// TwinCAT 3 PLC project PLC_LaserMarking_K2P3
// ProgramVersion: 3.1.4023.0
// libraries:
//   Tc2_MC2, * (Beckhoff Automation GmbH)
//   Tc2_Standard, * (Beckhoff Automation GmbH)
//   Tc2_System, * (Beckhoff Automation GmbH)
//   Tc3_MC2_AdvancedHoming, * (Beckhoff Automation GmbH)
//   Tc3_Module, * (Beckhoff Automation GmbH)
// project tree:
//   DUTs/ eAuto_State_Macine.TcTLEO, eLM_State_Machine.TcTLEO, eManual_State_Machine.TcTLEO, eMarking_Types.TcTLEO, eMC_State_Machine.TcTLEO, eUniquenessMethos.TcTLEO
//   GVLs/ GVL_AxisParameters.TcGVL, GVL_GateWay.TcGVL, GVL_IO.TcGVL, GVL_LaserMarking_MC_Parameters.TcGVL, GVL_StateMachine.TcGVL
//   / PlcTask.TcTTO
//   POUs/Alarms/ Alarm_Display_ST.TcPOU, Alarm_Flag.TcPOU, EtherCAT_Diagnostic.TcPOU
//   POUs/Main POUs/ Main.TcPOU, POU_GatewaySignals.TcPOU, POU_Manual_Auto.TcPOU, POU_Output.TcPOU
//   POUs/StateMachine_AutoManual/ AutoStates_POU.TcPOU
//   POUs/StateMachine_LaserMarking/ LaserMarking_Variable_Selection.TcPOU, LM_State_MC_TCP.TcPOU
//   POUs/StateMachine_MC_Axis/ MC_State_MC.TcPOU
// real-time tasks:
//   TASK PlcTask: cycle T#10ms, priority 20, ADS port 350
//   TASK PlcTask1: cycle T#10ms, priority 21, ADS port 351
// motion (NC):
//   TASK NC-Task SAF: cycle T#2ms, priority 4, ADS port 501
//   TASK NC-Task SVB: cycle T#10ms, priority 8, ADS port 511
//   AXIS Axis Y (id 2)
//     OtherSettings: AllowMotionCmdToSlave=true
//     encoder EncType=19
//       EncPara: MaxCount=#xffffffff
//     drive DrvType=16
//       DrvPara: MaxCount=#xffffffff, DriveControlDWord=#x00020000
//         Analog: TorqueScale=10, ScaleFactorActTorque=0.1
//         TimeComp: TaskDelayCycles=1
//     controller CtrType=1
//       CtrPara: PriorControlFactor=1
//         Observer: BandWidth=20
// I/O:
//   DEVICE Device 1 (EtherCAT), AmsNetId 192.168.0.10.2.1
//     Term 1 (EK1100) [EK1100 EtherCAT Coupler (2A E-Bus)]
//     Box 2 (ASDA-A2-E CoE Drive) [Delta ASDA-A2-E EtherCAT(CoE) Drive Rev4]
// variable links:
//   NC-Task SAF/Axes/Axis Y <-> Device 1 (EtherCAT)/Box 2 (ASDA-A2-E CoE Drive)
//     Drive/Inputs/In/nDcOutputTime <-> InfoData/DcOutputShift
//     Drive/Inputs/In/nState1 <-> 2nd TxPDO Mapping/Status Word
//     Drive/Inputs/In/nState2 <-> 2nd TxPDO Mapping/Status Word @bit 8
//     Drive/Inputs/In/nState4 @bit 1 <-> WcState/InputToggle
//     Drive/Inputs/In/nState4 <-> WcState/WcState
//     Drive/Outputs/Out/nCtrl1 <-> 2nd RxPDO Mapping/Control Word
//     Drive/Outputs/Out/nCtrl2 <-> 2nd RxPDO Mapping/Control Word @bit 8
//     Drive/Outputs/Out/nDataOut1 <-> 2nd RxPDO Mapping/TargetPosition
//     Enc/Inputs/In/nDataIn1 <-> 2nd TxPDO Mapping/ActualPosition
//     Enc/Inputs/In/nDcInputTime <-> InfoData/DcInputShift
//     Enc/Inputs/In/nState4 @bit 1 <-> WcState/InputToggle
//     Enc/Inputs/In/nState4 <-> WcState/WcState
//   PLC_LaserMarking_K2P3/PLC_LaserMarking_K2P3 Instance <-> NC-Task SAF/Axes/Axis Y
//     PlcTask Inputs/GVL_AxisParameters.YAxis.NcToPlc <-> Outputs/ToPlc
//     PlcTask Outputs/GVL_AxisParameters.YAxis.PlcToNc <-> Inputs/FromPlc

CONFIGURATION PLC_LaserMarking_K2P3
    RESOURCE PLC ON TwinCAT3
        TASK PlcTask(INTERVAL := T#10ms, PRIORITY := 21);
        PROGRAM Main WITH PlcTask : Main;
    END_RESOURCE
END_CONFIGURATION

// ---- DUTs/eAuto_State_Macine.TcTLEO
//{attribute 'qualified_only'}
{attribute 'strict'}
TYPE eAuto_State_Macine :
(
	Auto_Stop_State 	:= 0,
	Auto_Init_State 	:= 1,
	Auto_Ready_State 	:= 2,
	Auto_Y_Motion_State := 3,
	Auto_Marking_State 	:= 4
);
END_TYPE

// ---- DUTs/eLM_State_Machine.TcTLEO
//{attribute 'qualified_only'}
{attribute 'strict'}
TYPE eLM_State_Machine :
(
		LM_Off 			:= 0 ,
		LM_Init 		:= 1 ,
		LM_Ready 		:= 2 ,
		LM_CodeSend 	:= 3 ,
		LM_MarkCommand 	:= 4 ,
		LM_Feedback 	:= 5 
);
END_TYPE

// ---- DUTs/eManual_State_Machine.TcTLEO
//{attribute 'qualified_only'}
{attribute 'strict'}
TYPE eManual_State_Machine :
(
	Manual_Stop_State 	:= 0 ,
	Manual_Init_State 	:= 1 ,
	Manual_Ready_State 	:= 2 

);
END_TYPE

// ---- DUTs/eMarking_Types.TcTLEO
//{attribute 'qualified_only'}
{attribute 'strict'}
TYPE eMarking_Types :
(
		Plain_Text 		:= 0 ,
		DataMatrix_2D 	:= 1 ,
		QR_Code 		:= 2 ,
		BarCode 		:= 3 
);
END_TYPE

// ---- DUTs/eMC_State_Machine.TcTLEO
//{attribute 'qualified_only'}
{attribute 'strict'}
TYPE eMC_State_Machine :
(
		MC_Init 			:= 0 ,
		MC_Power 			:= 1 ,
		MC_Ready 			:= 2 ,
		MC_Home 			:= 3 ,
		MC_ManualMovement 	:= 4 ,
		MC_AutoMovement 	:= 5 ,
		MC_Error 			:= 6 ,
		MC_Reset 			:= 7

);
END_TYPE

// ---- DUTs/eUniquenessMethos.TcTLEO
//{attribute 'qualified_only'}
{attribute 'strict'}
TYPE eUniquenessMethos :
(
		PartCode 				:= 0 ,  //Machine ID and Partcode from Machine, Date and Time from PC
		PartCode_DateTime 		:= 1 ,  //Machine ID, Partcode,Date time from Machine. nothing from PC
		PartCode_LPC 			:= 2 ,  //Machine ID, Lifelong Production Count from Machine (9 Digit)
		WorkOrderNo_QtyCount	:= 3    //ERP WO Number with it's Qty count

);
END_TYPE

// ---- GVLs/GVL_AxisParameters.TcGVL
//{attribute 'qualified_only'}
VAR_GLOBAL
	YAxisAutoSpeed  		:  	LREAL;    			//
	YAxisManualSpeed  		:  	LREAL;    			//
	YAxisManualStep  		:  	BOOL := FALSE;    	//Step vise movement in Manual Mode
	YAxisManualStepDistFwd 	:  	LREAL := 100;    	//Distance to move in Step mode Forward Movement
	YAxisManualStepDistRev 	:  	LREAL := -100;    	//Distance to move in Step mode Reverse Movement
	YAxisAcceleration  		:  	LREAL := 100;    	//
	YAxisDeceleration  		:  	LREAL := 100;    	//
	YAxisEmgDeceleration  	:	LREAL := 1000; 	   	//
	YAxisJerk  :  LREAL 	:= 	100;    			//
	YAxisResetOnStop  		:	BOOL := TRUE;    	//

	YAxis 					:	AXIS_REF;			// 
	fbMC_Power				: 	MC_Power;			// Axis Power	
	fbMC_Reset				: 	MC_Reset;
	fbMC_Jog				:	MC_Jog;
	fbMC_Home				:	MC_Home;
	fbMC_MoveAbs			: 	MC_MoveAbsolute;
END_VAR

// ---- GVLs/GVL_GateWay.TcGVL
//{attribute 'qualified_only'}
VAR_GLOBAL

//*********INPUT Data ***********

ABS_IN_Marking_Command_IX100 	AT%IX10.0  	:  BOOL;    	//AnyBus card Command For start marking 
ABS_IN_EMERGENCY_IX101 			AT%IX10.1  	:  BOOL;    	//AnyBus card has received emergency signal
ABS_IN_OutPut_Type_IB00 		AT%IW0  	:  INT;    		//Anybus Type of Output on Conveypor
ABS_IN_Machine_ID_IB01 			AT%IW10  	:  STRING[15] := 'Godrej Mark'; 	//AnyBus Machine ID
ABS_IN_PartName_IW00 			AT%IW100  	:  STRING[15] := 'Default Value'; 	//Anybus Name Of Part
ABS_IN_Cordinate_1_ID00		 	AT%ID0  	:  REAL;    	//Anybus Y Cordinate 1
ABS_IN_Cordinate_2_ID10 		AT%ID1  	:  REAL;    	//Anybus Y Cordinate 2
ABS_IN_Cordinate_3_ID20 		AT%ID2  	:  REAL;    	//Anybus Y Cordinate 3
ABS_IN_Cordinate_4_ID30 		AT%ID3  	:  REAL;    	//Anybus Y Cordinate 4

//*********OUTPUT Data ***********

ABS_Out_Mark_Done_QX100 		AT%QX10.0  	:  BOOL;    	//Anybus Output for Marking Completed 
ABS_Out_EMG_Stop_QX101 			AT%QX10.1  	:  BOOL;    	//AnyBus Output for Gantry Emergency stop
ABS_Out_Machine_Healthy_QX102 	AT%QX10.2  	:  BOOL;    	//Anybus Output for Machinein healthy and operating condition
ABS_Out_Printing_data_Ok_QX103 	AT%QX10.3  	:  BOOL;    	//AnyBus Output for Printing Data OK


END_VAR

// ---- GVLs/GVL_IO.TcGVL
//{attribute 'qualified_only'}
VAR_GLOBAL


//*********INPUT MODULE EL1809 -1 ***********

Start_PB_IX00  			AT%IX0.0  :  BOOL;    //Start Push Button
Stop_PB_IX01  			AT%IX0.1  :  BOOL;    //Stop Push Button
Emg_PB_IX02 			AT%IX0.2  :  BOOL;    //Emergency Stop Push Button
AutoMan_SelSw_IX03 		AT%IX0.3  :  BOOL;    //Auto / Manual Selector Switch
FwdMotion_SelSw_IX04	AT%IX0.4  :  BOOL;    //Forward Selector Switch
RevMotion_SelSw_IX05 	AT%IX0.5  :  BOOL;    //Reverse Selector Switch
LaserOn_PB_IX06 		AT%IX0.6  :  BOOL;    //Laser ON
FwdLimit_Prxy_IX07 		AT%IX0.7  :  BOOL;    //Forward Limit Proxy

RevLimit_Prxy_IX10 		AT%IX1.0  :  BOOL;    //Reverse Limit / Home Proxy


//*********OUTPUT MODULE EL2809 -1 ***********

Start_PBLamp_QX00 		AT%QX0.0  :  BOOL;    //Start Push Button (IX0.0) Light
LaserOn_PBLamp_QX01 	AT%QX0.1  :  BOOL;    //Laser ON Push Button (IX0.6) Light
Red_TwrLamp_QX02 		AT%QX0.2  :  BOOL;    //Tower Lamp - Red Light
Green_TwrLamp_QX03 		AT%QX0.3  :  BOOL;    //Tower Lamp - Green Light
Amber_TwrLamp_QX04 		AT%QX0.4  :  BOOL;    //Tower Lamp - Amber Light




END_VAR

// ---- GVLs/GVL_LaserMarking_MC_Parameters.TcGVL
//{attribute 'qualified_only'}

VAR_GLOBAL CONSTANT

//Master Parameters

LM_MachineID  			:  UINT := 1;    					//
END_VAR

VAR_GLOBAL
LM_Type  				:  eMarking_Types := DataMatrix_2D;	//Type of Value to Mark
LM_UniqueTec  			:  eUniquenessMethos := PartCode; 	//Uniqueness Method


//Connection Parameters

LM_Con_IP_Hostname  	:  BOOL := FALSE;    				//0- IP address, 1-HostName
LM_IP_Adr  				:  STRING[256] := '172.26.1.181';  	//Laser Marking PC IP Address
LM_HostName  			:  STRING[256] := 'FBPC19I0001';  	//Laser Marking PC Hostname Address
LM_SourceIP_Port  		:  UINT := 9812;    				//Beckhoff PLC Port
LM_DestinationIP_Port  	:  UINT := 9812;    				//Destination PC Port

LM_Connection_Error  	:  BOOL := TRUE;    //Connection With Laser marking PC Broken
LM_Con_Rcv_TimeOutTime  :  UINT := 10;    	//Laser Machine post marking request, time allowed for timeout
LM_Con_Rcv_Size_Data  	:  UINT := 100;    	//Size of Data to receive
LM_Con_Ready  			:  BOOL;    		//LM Ready State Machine is Ready without any errors

//Marking Values 

LM_Marking_String  		:  STRING[32] := 'GODREJ MACHINE ID, PARTNAME';    //
LM_WorkOrder_No  		:  STRING[32] := 'PLN00000';    	//
END_VAR

VAR_GLOBAL RETAIN
LM_Production_Count  	:  ULINT;    						//Long_Production_Count
LM_WorkOrder_Qty_Instance  :  UINT := 1;    				//
END_VAR

VAR_GLOBAL
// Command Structure

LM_CodeSelection_Enable  	:  BOOL := FALSE;    //If Enable, different different codes can be selected by resetting code selection done bit. if disabled initial value to be contant 
LM_CodeSelection_Done  		:  BOOL := TRUE;    //If Code selection Enabled, required for resetting current coding method
LM_ArrCodeType  			:  ARRAY[0..1] OF BYTE := [16#31, 16#5F];    //Code Type Selection Command String to Send (Default walue 1_ in ASCII)
LM_ArrCodeTypeSize  		:  UINT := 2;    //Size of Code Selection Data
LM_ArrUniqueVal  			:  ARRAY[0..31] OF BYTE := [16#47, 16#4F, 16#44, 16#52, 16#45, 16#4A, 16#20, 16#44, 16#45, 16#46, 16#41, 16#55, 16#4C, 16#54, 16#20, 16#56, 16#41, 16#4C, 16#55, 16#45, 12(16#0)];    //Unique Value As per Type of Uniqueness Method selected (Default Value : 'GODREJ DEFAULT VALUE' in ASCII)
LM_ArrUniqueValSize  		:  UINT := 25;    //Size of Unique Value
LM_ArrMarkCmd  				:  ARRAY[0..1] OF BYTE := [16#5F, 16#4D];    //Marking Command String to send (Default Value _M in ASCII)
LM_ArrMarkCmdSize  			:  UINT := 2;    //Size of Marking Command


END_VAR

// ---- GVLs/GVL_StateMachine.TcGVL
//{attribute 'qualified_only'}
VAR_GLOBAL

//*********Machine Status Variables ***********

Machine_Auto  :  BOOL;    //System is Operating in Auto Mode
Machine_Manual  :  BOOL;    //System is Operating in Auto mode
Machine_Stop  :  BOOL;    //System is in Stop Mode

//*********State Machine Status Variables ***********

Auto_State_Macine  		:  eAuto_State_Macine := Auto_Stop_State;    		//Auto State Machine
Manual_State_Machine  	:  eManual_State_Machine := Manual_Stop_State;    	//Manual State Machine
MC_State_Machine  		:  eMC_State_Machine := MC_Reset;    				//MC1 State Machine
LM_State  				:  eLM_State_Machine := LM_Off;    					//Laser Marking TCP Communication State Machine

//********* MC Status Variables ***********

MC_Ready  			:  BOOL := FALSE;    //MC_State machine is On, and Ready without errors.
MC_Home_Done  		:  BOOL := FALSE;    //MC_HOME is Done, no need to do again
MC_MoveMentDone  	:  BOOL := FALSE;    //Done Requested Movement for this NMC

//********* Laser Machine Status Variables ***********

LM_PrintDataSent  	:  BOOL := FALSE;    //Data to Mark has been sent. mark command pending
LM_PrintCmdSent  	:  BOOL := FALSE;    //Mark Command has been sent. Feedback Pending

END_VAR

// ---- POUs/Main POUs/Main.TcPOU
PROGRAM Main
VAR
END_VAR

//Main POU Folder
POU_GatewaySignals();
POU_Manual_Auto();
POU_Output();

//Alarms Folder
Alarm_Display_ST();
Alarm_Display_ST();
EtherCAT_Diagnostic();

//StateMachine_AutoManual Folder
AutoStates_POU();

//StateMachine_MC_Axis Folder
MC_State_MC();

//StateMachine_LaserMarking Folder
LaserMarking_Variable_Selection();
LM_State_MC_TCP();

END_PROGRAM

// ---- POUs/Main POUs/POU_GatewaySignals.TcPOU
PROGRAM POU_GatewaySignals
VAR
END_VAR

// NETWORK 1

END_PROGRAM

// ---- POUs/Main POUs/POU_Manual_Auto.TcPOU
PROGRAM POU_Manual_Auto
VAR
END_VAR

// NETWORK 1

END_PROGRAM

// ---- POUs/Main POUs/POU_Output.TcPOU
PROGRAM POU_Output
VAR
END_VAR
//tower Lamp POU

// NETWORK 1

END_PROGRAM

// ---- POUs/Alarms/Alarm_Display_ST.TcPOU
PROGRAM Alarm_Display_ST
VAR
END_VAR

END_PROGRAM

// ---- POUs/Alarms/EtherCAT_Diagnostic.TcPOU
PROGRAM EtherCAT_Diagnostic
VAR
END_VAR

END_PROGRAM

// ---- POUs/StateMachine_AutoManual/AutoStates_POU.TcPOU
PROGRAM AutoStates_POU
VAR
END_VAR

END_PROGRAM

// ---- POUs/StateMachine_MC_Axis/MC_State_MC.TcPOU
PROGRAM MC_State_MC
VAR
END_VAR

//fbMC_Home.Options.ClearPositionLag := TRUE;
//fbMC_Home.Options.ReferenceMode;
//fbMC_Home.Options.SearchDirection;
//fbMC_Home.Options.SearchVelocity;
//fbMC_Home.Options.SyncDirection;
//fbMC_Home.Options.SyncVelocity;


Act_MotionAbsolute();
Act_MotionHome();
Act_MotionManual();
Act_MotionPower();
Act_MotionReset();

ACTION Act_MotionAbsolute:
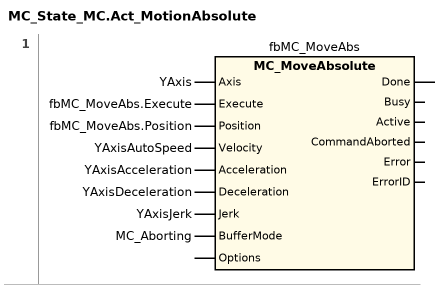
// NETWORK 1
fbMC_MoveAbs(
    Axis := YAxis,
    Execute := fbMC_MoveAbs.Execute,
    Position := fbMC_MoveAbs.Position,
    Velocity := YAxisAutoSpeed,
    Acceleration := YAxisAcceleration,
    Deceleration := YAxisDeceleration,
    Jerk := YAxisJerk,
    BufferMode := MC_Aborting); // MC_MoveAbsolute
END_ACTION

ACTION Act_MotionHome:
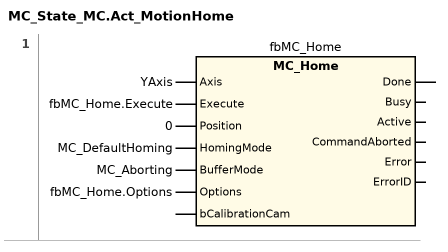
// NETWORK 1
fbMC_Home(
    Axis := YAxis,
    Execute := fbMC_Home.Execute,
    Position := 0,
    HomingMode := MC_DefaultHoming,
    BufferMode := MC_Aborting,
    Options := fbMC_Home.Options); // MC_Home
END_ACTION

ACTION Act_MotionManual:
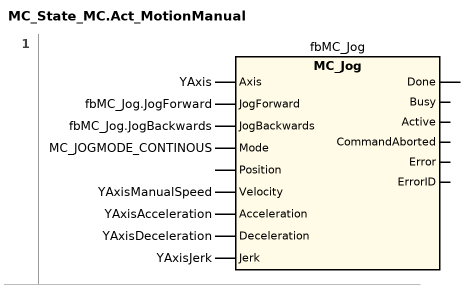
// NETWORK 1
fbMC_Jog(
    Axis := YAxis,
    JogForward := fbMC_Jog.JogForward,
    JogBackwards := fbMC_Jog.JogBackwards,
    Mode := MC_JOGMODE_CONTINOUS,
    Velocity := YAxisManualSpeed,
    Acceleration := YAxisAcceleration,
    Deceleration := YAxisDeceleration,
    Jerk := YAxisJerk); // MC_Jog
END_ACTION

ACTION Act_MotionPower:
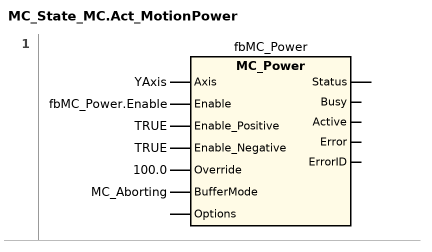
// NETWORK 1
fbMC_Power(
    Axis := YAxis,
    Enable := fbMC_Power.Enable,
    Enable_Positive := TRUE,
    Enable_Negative := TRUE,
    Override := 100.0,
    BufferMode := MC_Aborting); // MC_Power
END_ACTION

ACTION Act_MotionReset:
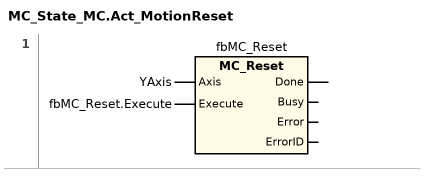
// NETWORK 1
fbMC_Reset(Axis := YAxis, Execute := fbMC_Reset.Execute); // MC_Reset
END_ACTION

END_PROGRAM

// ---- POUs/StateMachine_LaserMarking/LaserMarking_Variable_Selection.TcPOU
PROGRAM LaserMarking_Variable_Selection
VAR
END_VAR

END_PROGRAM

// ---- POUs/StateMachine_LaserMarking/LM_State_MC_TCP.TcPOU
PROGRAM LM_State_MC_TCP
VAR
END_VAR

// NETWORK 1

END_PROGRAM

// ---- POUs/Alarms/Alarm_Flag.TcPOU
PROGRAM Alarm_Flag
VAR
END_VAR

// NETWORK 1

END_PROGRAM
